Staubli VAL3: openGripper.pgx

program openGripper()
begin
  switchGripper=false
  message="openGripper:done"
  taskCreate "sendStatus",100,sendStatus()
  taskKill("openGripper")
end
